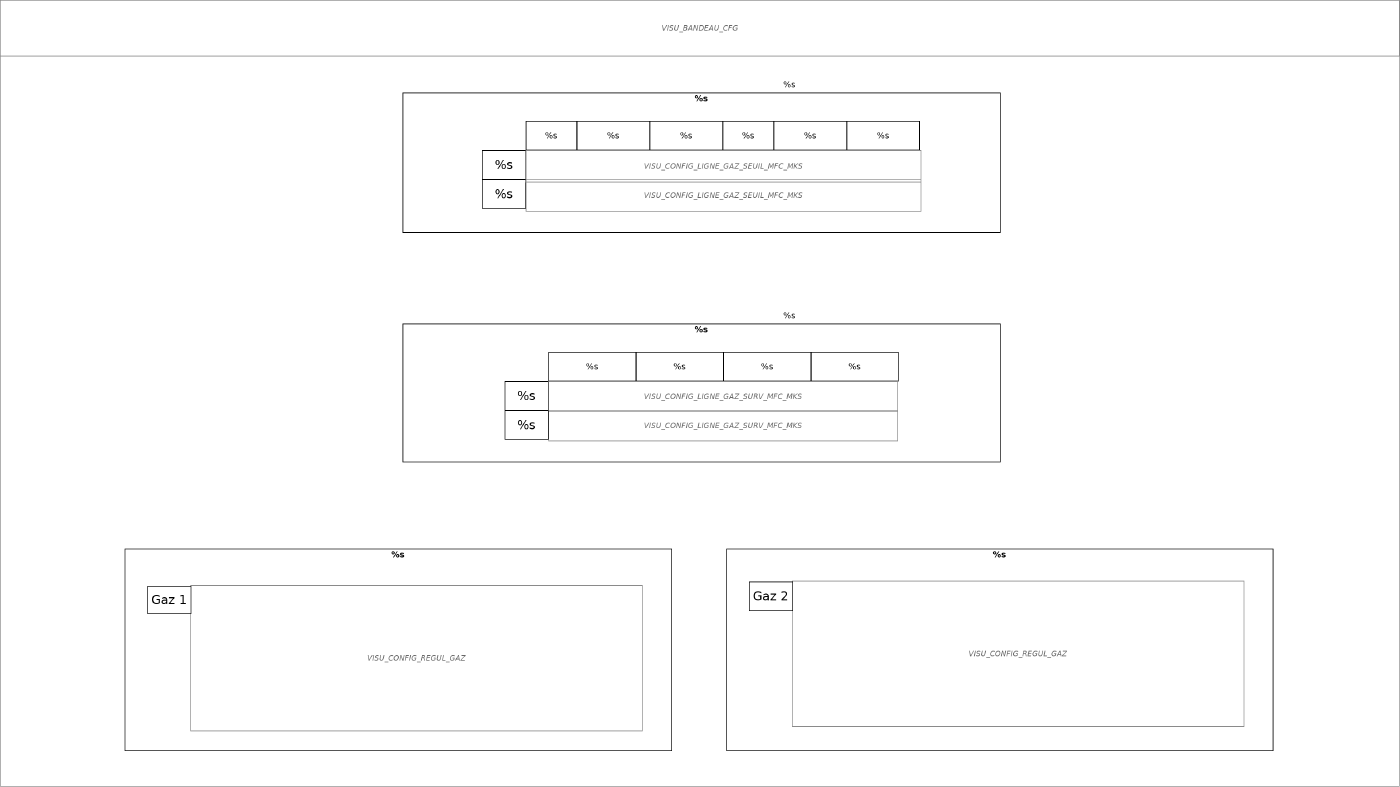
VISUALIZATION VISU_CONFIG_GAZ  // 1920x1080
    RoundedRectangle (996,753 750x277), "%s", text list: 'TextList_Config_Gaz', text index: 35
    RoundedRectangle (171,753 750x277), "%s", text list: 'TextList_Config_Gaz', text index: 35
    Frame (0,0 1920x77)
        shows VISU_BANDEAU_CFG()
    Frame (722,206 542x44)
        shows VISU_CONFIG_LIGNE_GAZ_SEUIL_MFC_MKS(m_Input_MASSFLOW := PRG_GAZ.DG[1])
    RoundedRectangle (552,127 820x192), "%s", text list: 'TextList_Config_Gaz', text index: 1
    Rectangle (1071,106 300x20), "%s", text list: 'TextList_Config_Gaz', text index: 3
    Rectangle (1071,423 300x20), "%s", text list: 'TextList_Config_Gaz', text index: 4
    RoundedRectangle (552,444 820x190), "%s", text list: 'TextList_Config_Gaz', text index: 2
    Rectangle (791,166 100x40), "%s", text list: 'TextList_Config_Gaz', text index: 6
    Rectangle (891,166 100x40), "%s", text list: 'TextList_Config_Gaz', text index: 7
    Rectangle (1161,166 100x40), "%s", text list: 'TextList_Config_Gaz', text index: 9
    Rectangle (991,166 70x40), "%s", text list: 'TextList_Config_Gaz', text index: 8
    Rectangle (1061,166 100x40), "%s", text list: 'TextList_Config_Gaz', text index: 6
    Rectangle (721,166 70x40), "%s", text list: 'TextList_Config_Gaz', text index: 5
    Rectangle (661,206 60x40), "%s", text list: 'TextList_Config_Gaz', text index: 11
    Frame (721,246 542x44)
        shows VISU_CONFIG_LIGNE_GAZ_SEUIL_MFC_MKS(m_Input_MASSFLOW := PRG_GAZ.DG[2])
    Rectangle (661,246 60x40), "%s", text list: 'TextList_Config_Gaz', text index: 12
    Frame (721,206 542x44)
        shows VISU_CONFIG_LIGNE_GAZ_SEUIL_MFC_MKS(m_Input_MASSFLOW := PRG_GAZ.DG[1])
        p1532468285: PRG_GAZ.DG[1]
    Rectangle (692,523 60x40), "%s", text list: 'TextList_Config_Gaz', text index: 11
    Rectangle (1112,483 120x40), "%s", text list: 'TextList_Config_Gaz', text index: 23
    Rectangle (872,483 120x40), "%s", text list: 'TextList_Config_Gaz', text index: 21
    Rectangle (992,483 120x40), "%s", text list: 'TextList_Config_Gaz', text index: 22
    Rectangle (752,483 120x40), "%s", text list: 'TextList_Config_Gaz', text index: 20
    Frame (752,523 479x42)
        shows VISU_CONFIG_LIGNE_GAZ_SURV_MFC_MKS(m_Input_MASSFLOW := PRG_GAZ.DG[1])
    Frame (752,563 479x42)
        shows VISU_CONFIG_LIGNE_GAZ_SURV_MFC_MKS(m_Input_MASSFLOW := PRG_GAZ.DG[2])
    Rectangle (692,563 60x40), "%s", text list: 'TextList_Config_Gaz', text index: 12
    Frame (261,803 620x200)
        shows VISU_CONFIG_REGUL_GAZ(m_Input_REGULATION := Global_Variables.PRG_GAZ.REGULATION_GAZ_L1)
    Rectangle (202,804 60x38), "Gaz 1"
    Frame (1086,797 620x200)
        shows VISU_CONFIG_REGUL_GAZ(m_Input_REGULATION := Global_Variables.PRG_GAZ.REGULATION_GAZ_L2)
    Rectangle (1027,798 60x40), "Gaz 2"
END_VISUALIZATION

(* stored: Version 1.1.0.1, ProductVersion 3.1.4024.12
   Visu VISU_CONFIG_GAZ: Id {d5b2d709-1415-4c45-982d-28519bd087ae} *)
